// TIA Portal V21 export
TYPE "Std_stTimer"
   STRUCT
      IN : Bool;   // Avvio Conteggio
      O : Bool;   // Fine Conteggio
      Preset : Real;   // Durata Del Ritardo All'Inserzione
      TempoTrascorso : Real;   // Valore Temporale Attuale
   END_STRUCT;
END_TYPE
